{attribute 'linkalways'} 
{attribute 'no_explicit_call' := 'This FB is a CLASS and must be accessed using methods or properties'}
{attribute 'enable_dynamic_creation'}
FUNCTION_BLOCK Node_F_VN_GetImageHeight EXTENDS VisionNode
VAR
    ipImage : _ITcVnImage;
    nHeight : _UDINT(0);
    hrPrev : _HRESULT(S_OK);
	hresult : _HRESULT(S_OK);
END_VAR

METHOD PUBLIC  Clone : I_Node
VAR
	pNode : POINTER TO Node_F_VN_GetImageHeight;
END_VAR
pNode := __NEW(Node_F_VN_GetImageHeight);
Clone := pNode^;
END_METHOD

METHOD FB_init : BOOL
VAR_INPUT
	bInitRetains : BOOL; // if TRUE, the retain variables are initialized (warm start / cold start)
	bInCopyCode : BOOL;  // if TRUE, the instance afterwards gets moved into the copy code (online change)
END_VAR
AddInput('ipImage', ipImage);
AddInput('hrPrev', hrPrev);
AddOutput('nHeight', nHeight);
AddOutput('hresult', hresult);
END_METHOD

METHOD PROTECTED OnExecute : HRESULT
hresult.Value := F_VN_GetImageHeight(
    ipImage := ipImage.Value,
    nHeight := nHeight.Value,
	hrPrev:= hrPrev.Value);
END_METHOD

METHOD PUBLIC PreExecutionCheck
VAR_INPUT
	Check : I_PreExecutionChecks;
END_VAR
IF FAILED(hrPrev.Value) THEN
    RETURN;
END_IF

Check.IsTrue(ipImage.IsValid, 'ipImage must contain an image');
END_METHOD

END_FUNCTION_BLOCK

(* stored: Version 1.1.0.1, ProductVersion 3.1.4024.13
   POU Node_F_VN_GetImageHeight: Id {8539a53d-68b7-0c6d-2c7a-bcef40622d24}, SpecialFunc None
   Folder Constructor: Id {95726090-40ea-0529-25d9-82a91919937f}
   Method Clone: Id {861c7af2-1500-081c-180f-4bd4975d7a2b}
   Method FB_init: Id {1d1ee0ef-4c4c-02f3-1f77-d4293be5c56d}
   Method OnExecute: Id {7e14b4e5-c403-0629-249b-e8ea4dd49532}
   Method PreExecutionCheck: Id {f74baa13-1f3a-07bd-233a-2af596124661} *)
